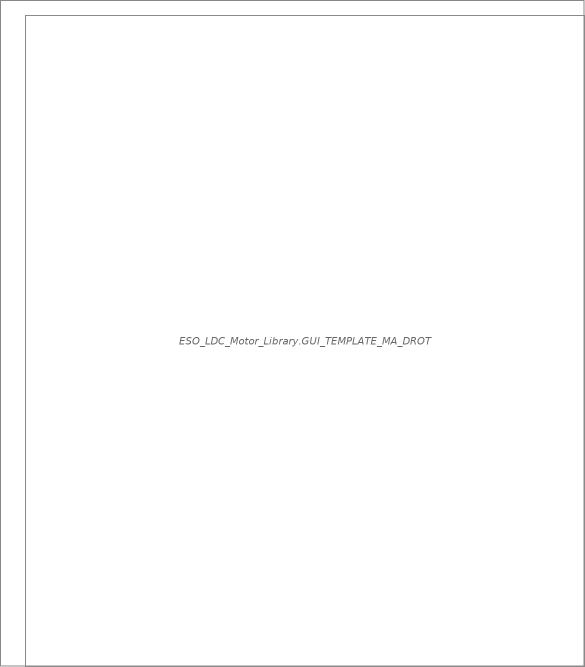
VISUALIZATION drot1  // 585x667
    Frame (25,15 560x652)
        shows ESO_LDC_Motor_Library.GUI_TEMPLATE_MA_DROT(m_DeviceName := 'drot1', m_Instance := MAIN.drot1)
END_VISUALIZATION

(* stored: Version 1.1.0.1, ProductVersion 3.1.4024.3
   Visu drot1: Id {2bf90a6f-c7c0-43c9-8884-e7eea155e75b} *)
